TYPE ST_Message :
STRUCT
	eLogLevel:			E_LogLevel;
	nID:				UDINT;
	nTimestamp:			ULINT;	
	sSource:			STRING(255);
	sMessage:			STRING(255);
	sDefault:			STRING(255);
	sArguments:			STRING(255);
	bActive:			BOOL;
END_STRUCT
END_TYPE

(* stored: Version 1.1.0.1
   DUT ST_Message: Id {56bff33d-8470-42da-bea5-9559cbe6e709} *)
